FUNCTION_BLOCK Seguridad
VAR_INPUT
	
	CuadroPrincipalRunStop AT%I*:BOOL;
	CuadroPrincipalAutomatico AT%I*:BOOL;
	SeguridadSetas AT%I*:BOOL;
END_VAR
VAR_OUTPUT
	CuadroLedVerde AT%Q*:BOOL;
	CuadroLedAmarillo AT%Q*:BOOL;
	
	MotorSuperior_Freq  AT%Q*: UINT;
	MotorSuperior_Command AT%Q*: INT;
		
	MotorInferior_Freq  AT%Q*: UINT;
	MotorInferior_Command AT%Q*: INT;
	
	LineaReady :BOOL;
	FinTiempoTON :TON;
	
	
	
END_VAR
VAR
	FlancoRunStop:R_TRIG;
	TempCiclo:TON;
	TempRetraso:TON;
	Resultados : ResultadoCiclo;

	puesto: INT;
	Falso: BOOL;
END_VAR

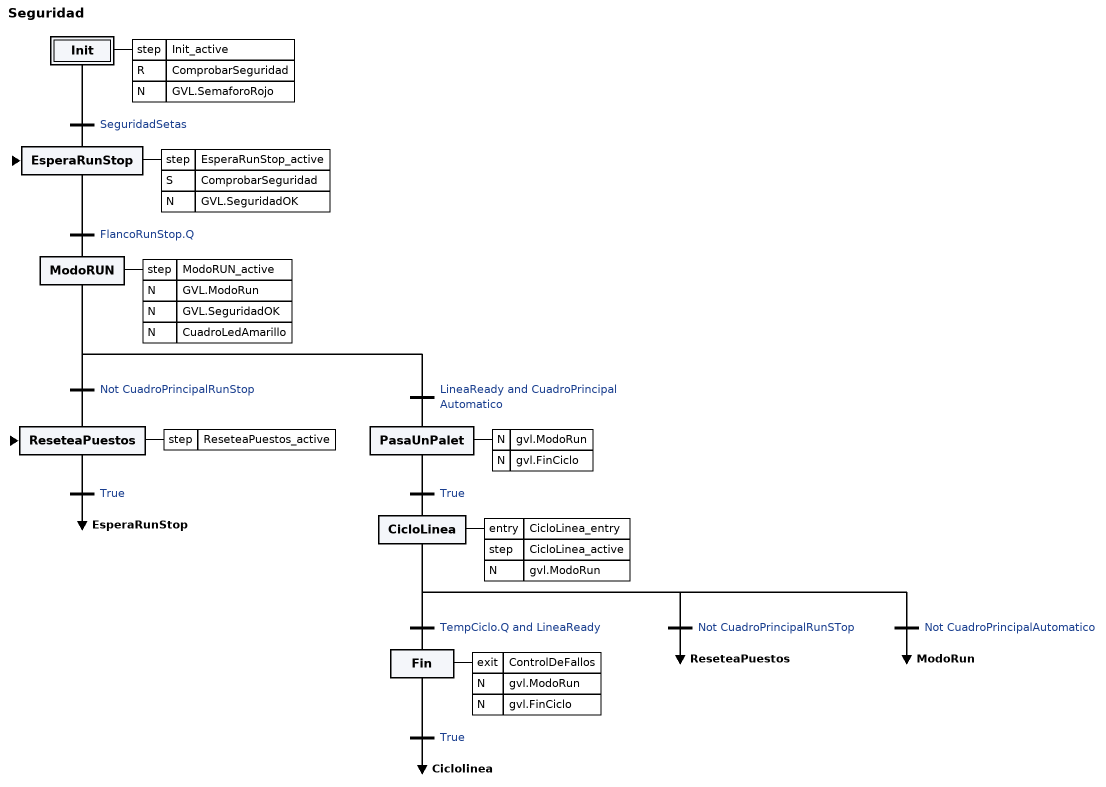
INITIAL_STEP Init:
    Init_active(N);  // step action
    ComprobarSeguridad(R);
    GVL.SemaforoRojo(N);
END_STEP
TRANSITION FROM Init TO EsperaRunStop
    := SeguridadSetas;
END_TRANSITION
STEP EsperaRunStop:  // min time T#1s
    EsperaRunStop_active(N);  // step action
    ComprobarSeguridad(S);
    GVL.SeguridadOK(N);
END_STEP
TRANSITION FROM EsperaRunStop TO ModoRUN
    := FlancoRunStop.Q;
END_TRANSITION
STEP ModoRUN:  // min time T#1s
    ModoRUN_active(N);  // step action
    GVL.ModoRun(N);
    GVL.SeguridadOK(N);
    CuadroLedAmarillo(N);
END_STEP
TRANSITION FROM ModoRUN TO ReseteaPuestos
    := Not CuadroPrincipalRunStop;
END_TRANSITION
STEP ReseteaPuestos:  // min time T#1s
    ReseteaPuestos_active(N);  // step action
END_STEP
TRANSITION FROM ReseteaPuestos TO EsperaRunStop
    := True;
END_TRANSITION
TRANSITION FROM ModoRUN TO PasaUnPalet
    := LineaReady and CuadroPrincipalAutomatico;
END_TRANSITION
STEP PasaUnPalet:  // min time T#3s
    gvl.ModoRun(N);
    gvl.FinCiclo(N);
END_STEP
TRANSITION FROM PasaUnPalet TO CicloLinea
    := True;
END_TRANSITION
STEP CicloLinea:  // min time T#4s
    CicloLinea_entry(P1);  // entry action
    CicloLinea_active(N);  // step action
    gvl.ModoRun(N);
END_STEP
TRANSITION FROM CicloLinea TO Fin
    := TempCiclo.Q and LineaReady;
END_TRANSITION
STEP Fin:  // min time T#3s
    ControlDeFallos(P0);  // exit action
    gvl.ModoRun(N);
    gvl.FinCiclo(N);
END_STEP
TRANSITION FROM Fin TO Ciclolinea
    := True;
END_TRANSITION
TRANSITION FROM CicloLinea TO ReseteaPuestos
    := Not CuadroPrincipalRunSTop;
END_TRANSITION
TRANSITION FROM CicloLinea TO ModoRun
    := Not CuadroPrincipalAutomatico;
END_TRANSITION

ACTION CicloLinea_active:
TempCiclo(IN:=TRUE);
TempRetraso(IN:=TempCiclo.Q);

gvl.SemaforoVerde := TRUE;

IF (    (ElevadorInicioLinea.Ready OR gvl.ModoDobleCarga)///no esperamos por elevador inicio en modo doble carga
	AND (ElevadorFinLinea.ready OR GVL.Puesto92.EsperandoPalet ) //si el ultimo  puesto no tieen palet no esperamos por elevador fin
	AND GVL.Puesto11.FinPuesto AND
		GVL.Puesto12.FinPuesto AND
		GVL.Puesto21.FinPuesto AND
		GVL.Puesto22.FinPuesto AND
		GVL.Puesto31.FinPuesto AND
		GVL.Puesto32.FinPuesto AND
		GVL.Puesto41.FinPuesto AND
		GVL.Puesto42.FinPuesto AND
		GVL.Puesto51.FinPuesto AND
		GVL.Puesto52.FinPuesto AND
		GVL.Puesto61.FinPuesto AND
		GVL.Puesto62.FinPuesto AND
		GVL.Puesto71.FinPuesto AND
		GVL.Puesto72.FinPuesto AND
		GVL.Puesto81.FinPuesto AND
		GVL.Puesto82.FinPuesto AND
		GVL.Puesto91.FinPuesto AND
		(gvl.Puesto81.LuzRoja = FALSE) AND
		(GVL.Puesto92.FinPuesto OR gvl.ModoDobleCarga))
THEN
		LineaReady := TRUE;
		gvl.SemaforoAmarillo :=  FALSE;
ELSE 
	    LineaReady := FALSE;
		gvl.SemaforoAmarillo := TempCiclo.Q;
END_IF


IF TempCiclo.Q AND NOT Lineaready THEN

		IF NOT  GVL.Puesto11.FinPuesto THEN gvl.Est_Resultados[gvl.PunteroEst].RetrasoPuesto[1] := TIME_TO_INT(TempRetraso.ET)/1000; END_IF 
		IF NOT 	GVL.Puesto12.FinPuesto THEN gvl.Est_Resultados[gvl.PunteroEst].RetrasoPuesto[2] := TIME_TO_INT(TempRetraso.ET); END_IF 
		if not 	GVL.Puesto21.FinPuesto then gvl.Est_Resultados[gvl.PunteroEst].RetrasoPuesto[3] := TIME_TO_INT(TempRetraso.ET); END_IF 
		if not 	GVL.Puesto22.FinPuesto then gvl.Est_Resultados[gvl.PunteroEst].RetrasoPuesto[4] := TIME_TO_INT(TempRetraso.ET); END_IF 
		if not 	GVL.Puesto31.FinPuesto then gvl.Est_Resultados[gvl.PunteroEst].RetrasoPuesto[5] := TIME_TO_INT(TempRetraso.ET); END_IF 
		if not 	GVL.Puesto32.FinPuesto then gvl.Est_Resultados[gvl.PunteroEst].RetrasoPuesto[6] := TIME_TO_INT(TempRetraso.ET); END_IF 
		if not 	GVL.Puesto41.FinPuesto then gvl.Est_Resultados[gvl.PunteroEst].RetrasoPuesto[7] := TIME_TO_INT(TempRetraso.ET); END_IF 
		if not 	GVL.Puesto42.FinPuesto then gvl.Est_Resultados[gvl.PunteroEst].RetrasoPuesto[8] := TIME_TO_INT(TempRetraso.ET); END_IF 
		if not 	GVL.Puesto51.FinPuesto then gvl.Est_Resultados[gvl.PunteroEst].RetrasoPuesto[9] := TIME_TO_INT(TempRetraso.ET); END_IF 
		if not 	GVL.Puesto52.FinPuesto then gvl.Est_Resultados[gvl.PunteroEst].RetrasoPuesto[10] := TIME_TO_INT(TempRetraso.ET); END_IF 
		if not 	GVL.Puesto61.FinPuesto then gvl.Est_Resultados[gvl.PunteroEst].RetrasoPuesto[11] := TIME_TO_INT(TempRetraso.ET); END_IF 
		if not 	GVL.Puesto62.FinPuesto then gvl.Est_Resultados[gvl.PunteroEst].RetrasoPuesto[12] := TIME_TO_INT(TempRetraso.ET); END_IF 
		if not 	GVL.Puesto71.FinPuesto then gvl.Est_Resultados[gvl.PunteroEst].RetrasoPuesto[13] := TIME_TO_INT(TempRetraso.ET); END_IF 
		if not 	GVL.Puesto72.FinPuesto then gvl.Est_Resultados[gvl.PunteroEst].RetrasoPuesto[14] := TIME_TO_INT(TempRetraso.ET); END_IF 
		if not 	GVL.Puesto81.FinPuesto then gvl.Est_Resultados[gvl.PunteroEst].RetrasoPuesto[15] := TIME_TO_INT(TempRetraso.ET); END_IF 
		if not 	GVL.Puesto82.FinPuesto then gvl.Est_Resultados[gvl.PunteroEst].RetrasoPuesto[16] := TIME_TO_INT(TempRetraso.ET); END_IF 
		if not 	GVL.Puesto91.FinPuesto then gvl.Est_Resultados[gvl.PunteroEst].RetrasoPuesto[17] := TIME_TO_INT(TempRetraso.ET); END_IF 
		if not 	GVL.Puesto92.FinPuesto then gvl.Est_Resultados[gvl.PunteroEst].RetrasoPuesto[18] := TIME_TO_INT(TempRetraso.ET); END_IF 

END_IF
END_ACTION

ACTION CicloLinea_entry:
TempCiclo(IN:=FALSE, PT:= DWORD_TO_TIME(  (INT_TO_DWORD(gvl.TiempoDeCiclo) -3)* 1000));
TempRetraso(IN:=FALSE, PT:= T#15M);



gvl.PunteroEst := gvl.PunteroEst +1;
IF gvl.PunteroEst > 1999 THEN
	gvl.PunteroEst := 1;
END_IF


//Creamos un nuevo registros
gvl.Est_Resultados[gvl.PunteroEst].Ciclo := gvl.TiempoDeCiclo;
gvl.Est_Resultados[gvl.PunteroEst].Producto := gvl.Producto;
gvl.Est_Resultados[gvl.PunteroEst].hora := gvl.HoraActual;



FOR puesto := 1 TO 18 DO
	gvl.Est_Resultados[gvl.PunteroEst].FalloPuesto[puesto] := FALSE;
	gvl.Est_Resultados[gvl.PunteroEst].RetrasoPuesto[puesto] := 0;
	
END_FOR
END_ACTION

ACTION ComprobarSeguridad:
IF NOT SeguridadSetas THEN
	SFCReset:=TRUE;
END_IF
END_ACTION

ACTION ControlDeFallos:




//avanzamos el fallo en el palet y guardamos estadistica
FOR puesto := 18 TO 2 BY -1 DO
	gvl.Est_Resultados[gvl.PunteroEst].FalloPuesto[puesto] := gvl.FalloPallet[puesto];
	gvl.FalloPallet[puesto] := gvl.FalloPallet[puesto -1 ];
END_FOR

gvl.FalloPallet[1] := Falso;
END_ACTION

ACTION EsperaRunStop_active:
FlancoRunStop(CLK:=CuadroPrincipalRunStop);

Gvl.SemaforoAmarillo := TRUE;
MotorCintaSuperior(0);
MotorCintaInferior(0);
END_ACTION

ACTION Init_active:
MotorCintaSuperior(0);
MotorCintaInferior(0);
SFCreset := FALSE;
gvl.SemaforoAmarillo :=FALSE;
gvl.SemaforoVerde := FALSE;
END_ACTION

ACTION ModoRUN_active:

TempCiclo(IN:=FALSE);

IF ElevadorFinLinea.Ready THEN
 MotorCintaSuperior(1);
END_IF

gvl.SemaforoAmarillo :=TRUE;

IF ElevadorInicioLinea.EsperandoPalet OR ElevadorInicioLinea.Ready THEN
	MotorCintaInferior(1);
END_IF

IF (ElevadorInicioLinea.Ready AND
	ElevadorFinLinea.ready AND 
	GVL.Puesto12.FinPuesto AND
	GVL.Puesto21.FinPuesto AND
	GVL.Puesto22.FinPuesto AND
	GVL.Puesto31.FinPuesto AND
	GVL.Puesto32.FinPuesto AND
	GVL.Puesto41.FinPuesto AND
	GVL.Puesto42.FinPuesto AND
	GVL.Puesto51.FinPuesto AND
	GVL.Puesto52.FinPuesto AND
	GVL.Puesto61.FinPuesto AND
	GVL.Puesto62.FinPuesto AND
	GVL.Puesto71.FinPuesto AND
	GVL.Puesto72.FinPuesto AND
	GVL.Puesto81.FinPuesto AND
	GVL.Puesto82.FinPuesto AND
	GVL.Puesto91.FinPuesto )
THEN		
		gvl.SemaforoVerde := TRUE;
		LineaReady := TRUE;
			
ELSE
			LineaReady:=FALSE;
			gvl.FinTiempo :=FALSE;
			gvl.SemaforoVerde := FALSE;
END_IF
END_ACTION

METHOD PRIVATE MotorCintaInferior : BOOL
VAR_INPUT
	Direccion: INT;
END_VAR
MotorInferior_Freq := gvl.VelocidadCinta * 100;


MotorInferior_Command := 0;
MotorInferior_Command.7 := 1 ; //Control Word Active


IF Direccion  = 0 THEN
	MotorInferior_Command.3 := 1 ; // Stop according to parameter setting	

ELSIF gvl.ElevadorInicioLinea.PresenciaCintaAbajo AND NOT gvl.ElevadorInicioLinea.SensorAbajo THEN
	// presencia en la salida y el elevador no esta abajo: paramos y ERROR
	MotorInferior_Command.3 := 1 ;
	
ELSIF Direccion  = 1 THEN		
		MotorInferior_Command.2 := 1 ; //1 reversed 0 fordward
		MotorInferior_Command.0 := 1 ; // Run Command active
ELSE
	MotorInferior_Command.3 := 1 ; // Stop according to parameter setting	
END_IF
END_METHOD

METHOD PRIVATE MotorCintaSuperior : BOOL
VAR_INPUT
	Direccion: INT;
END_VAR
MotorSuperior_Freq := gvl.VelocidadCinta * 100;


MotorSuperior_Command := 0;
MotorSuperior_Command.7 := 1 ; //Control Word Active

IF Direccion = 0 THEN
	MotorSuperior_Command.3 := 1 ; // Stop according to parameter setting	
ELSIF gvl.Elevadorfinlinea.PresenciaCintaArriba AND NOT gvl.Elevadorfinlinea.sensorarriba THEN
	//ERROR : palet en la salida y elevador no arriba
	MotorSuperior_Command.3 := 1 ;
ELSIF Direccion  = 1 THEN		
		MotorSuperior_Command.2 := 0 ; //1 reversed 0 fordward
		MotorSuperior_Command.0 := 1 ; // Run Command active
ELSE
	MotorSuperior_Command.3 := 1 ; // Stop according to parameter setting	
END_IF
END_METHOD

ACTION ReseteaPuestos_active:

//Resetea los puestos para pasar un palet


GVL.Puesto11.SFCreset := TRUE;
GVL.Puesto12.SFCreset := TRUE;
GVL.Puesto21.SFCreset := TRUE;
GVL.Puesto22.SFCreset := TRUE;
GVL.Puesto31.sfcreset := TRUE;
GVL.Puesto32.sfcreset := TRUE;
GVL.Puesto41.sfcreset := TRUE;
GVL.Puesto42.sfcreset := TRUE;
GVL.Puesto51.sfcreset := TRUE;
GVL.Puesto52.sfcreset := TRUE;
GVL.Puesto61.sfcreset := TRUE;
GVL.Puesto62.sfcreset := TRUE;
GVL.Puesto71.sfcreset := TRUE;
GVL.Puesto72.sfcreset := TRUE;
GVL.Puesto81.sfcreset := TRUE;
GVL.Puesto82.sfcreset := TRUE;
GVL.Puesto91.sfcreset := TRUE;
GVL.Puesto92.sfcreset := TRUE;

ElevadorInicioLinea.SFCreset := TRUE;
ElevadorFinLinea.SFCreset := TRUE;
END_ACTION

END_FUNCTION_BLOCK

(* stored: Version 1.1.0.1, ProductVersion 3.1.4024.3
   POU Seguridad: Id {4569f4ce-7c18-43b2-b6d2-c84b9b228987}, SpecialFunc None
   Action CicloLinea_active: Id {10c95d75-f399-4dc5-aae0-0b73a7f56992}
   Action CicloLinea_entry: Id {ba3e33f5-6fcf-45f5-9190-4764bf44691b}
   Action ComprobarSeguridad: Id {7bf695df-134b-461a-8076-612d34882cfb}
   Action ControlDeFallos: Id {31645b11-331d-4389-8c5f-6526e1dfd6bb}
   Action EsperaRunStop_active: Id {1403c2f3-23a7-41d2-8640-6c276ea6723a}
   Action Init_active: Id {92180a6b-d030-4817-b874-17e008391633}
   Action ModoRUN_active: Id {3d03e4c2-a57c-4164-b30e-07c18b64000b}
   Method MotorCintaInferior: Id {4dd83318-4905-46c4-8553-8aafc8299076}
   Method MotorCintaSuperior: Id {47a5a076-0660-42e6-aa83-a7b0e8c717a5}
   Action ReseteaPuestos_active: Id {62f95641-774b-4a26-8ab2-96e7f8af90ad} *)
